Omron CX-Programmer project NewProject (CX-Programmer 9.73)

# PLC NewPLC1: CP1L M

## Global symbols (name address type ; comment)
0.00 BOOL  ; caco
0.01 BOOL  ; box1
0.02 BOOL  ; box2
0.03 BOOL  ; box3
0.04 BOOL  ; box4
0.05 BOOL  ; box5
0.06 BOOL  ; box6
0.07 BOOL  ; reset contagem
0.08 BOOL  ; total peças
0.09 BOOL  ; seleção comercial
D0 CHANNEL  ; contagem box 0
D10 CHANNEL  ; contagem box 5
D12 CHANNEL  ; contagem box 6
D14 CHANNEL  ; contagem total
D18 CHANNEL  ; contador amostragem
D2 CHANNEL  ; contagem box 1
D4 CHANNEL  ; contagem box 2
D6 CHANNEL  ; contagem box 3
D630 CHANNEL  ; Segundos Relógio
D631 CHANNEL  ; Minutos relógio
D632 CHANNEL  ; Horas relógio
D633 CHANNEL  ; Dia relógio
D634 CHANNEL  ; Mes Relógio
D635 CHANNEL  ; Ano relógio
D700 CHANNEL  ; hora ihm
D7003 CHANNEL  ; hora envio
D701 CHANNEL  ; minuto da ihm
D702 CHANNEL  ; segundo ihm
D703 CHANNEL  ; hora do envio
D704 CHANNEL  ; minuto envio
D705 CHANNEL  ; segundo envio
D8 CHANNEL  ; contagem box 4
H10.00 BOOL  ; reset contador
H10.01 BOOL  ; envia relogio
ch400 400 CHANNEL

## Program NewProgram1 (cyclic task 0)
Local symbols
TIM 0.12 BOOL
bit2 BOOL
d400D400 CHANNEL

### Section Controle_Qualidade

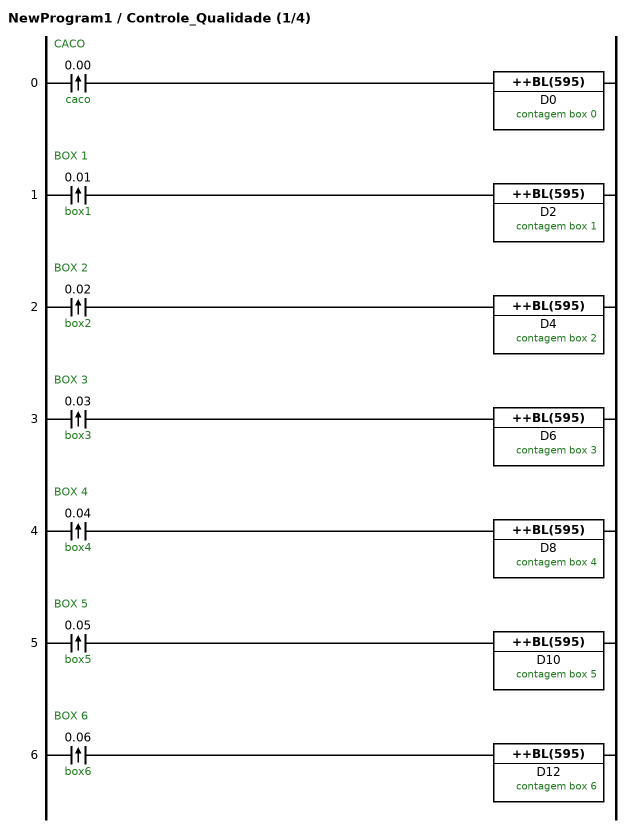
; rung 0: CACO
@LD 0.00  ; caco
++BL(595) D0  ; contagem box 0
; rung 1: BOX 1
@LD 0.01  ; box1
++BL(595) D2  ; contagem box 1
; rung 2: BOX 2
@LD 0.02  ; box2
++BL(595) D4  ; contagem box 2
; rung 3: BOX 3
@LD 0.03  ; box3
++BL(595) D6  ; contagem box 3
; rung 4: BOX 4
@LD 0.04  ; box4
++BL(595) D8  ; contagem box 4
; rung 5: BOX 5
@LD 0.05  ; box5
++BL(595) D10  ; contagem box 5
; rung 6: BOX 6
@LD 0.06  ; box6
++BL(595) D12  ; contagem box 6

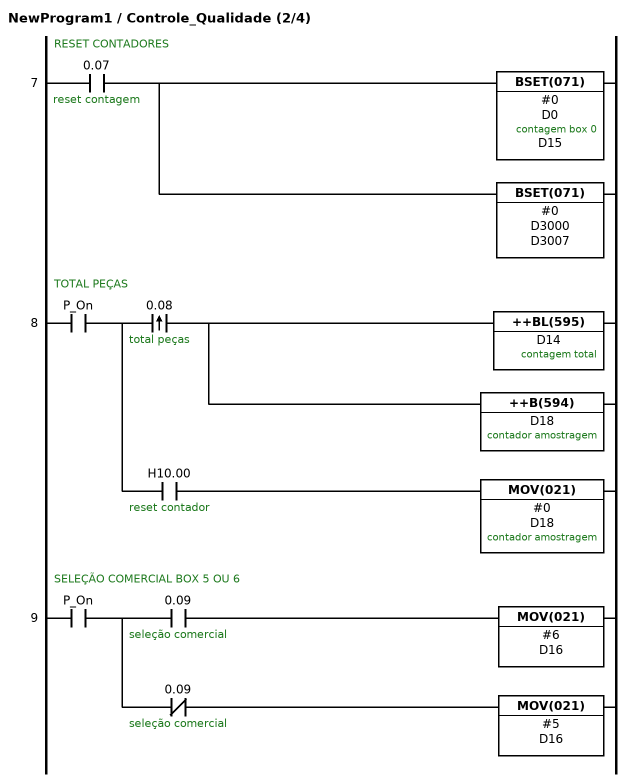
; rung 7: RESET CONTADORES
LD 0.07  ; reset contagem
BSET(071) #0 D0 D15  ; contagem box 0
BSET(071) #0 D3000 D3007
; rung 8: TOTAL PEÇAS
LD P_On
OUT TR0
@AND 0.08  ; total peças
++BL(595) D14  ; contagem total
++B(594) D18  ; contador amostragem
LD TR0
AND H10.00  ; reset contador
MOV(021) #0 D18  ; contador amostragem
; rung 9: SELEÇÃO COMERCIAL BOX 5 OU 6
LD P_On
OUT TR0
AND 0.09  ; seleção comercial
MOV(021) #6 D16
LD TR0
ANDNOT 0.09  ; seleção comercial
MOV(021) #5 D16

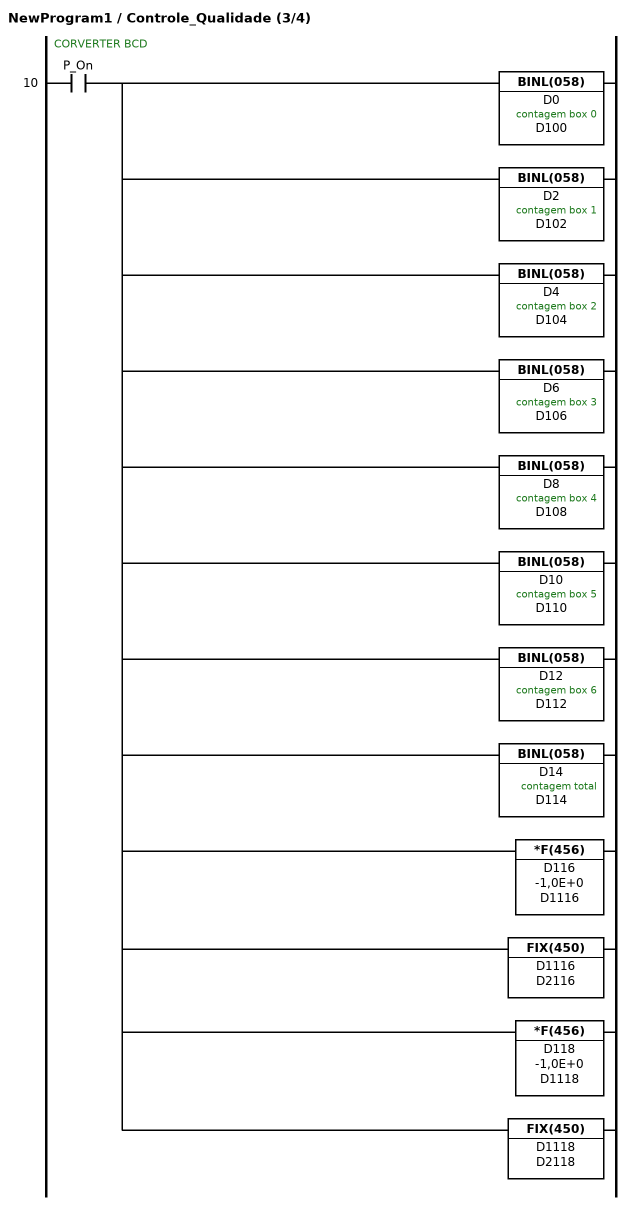
; rung 10: CORVERTER BCD
LD P_On
BINL(058) D0 D100  ; contagem box 0
BINL(058) D2 D102  ; contagem box 1
BINL(058) D4 D104  ; contagem box 2
BINL(058) D6 D106  ; contagem box 3
BINL(058) D8 D108  ; contagem box 4
BINL(058) D10 D110  ; contagem box 5
BINL(058) D12 D112  ; contagem box 6
BINL(058) D14 D114  ; contagem total
*F(456) D116 -1,0E+0 D1116
FIX(450) D1116 D2116
*F(456) D118 -1,0E+0 D1118
FIX(450) D1118 D2118

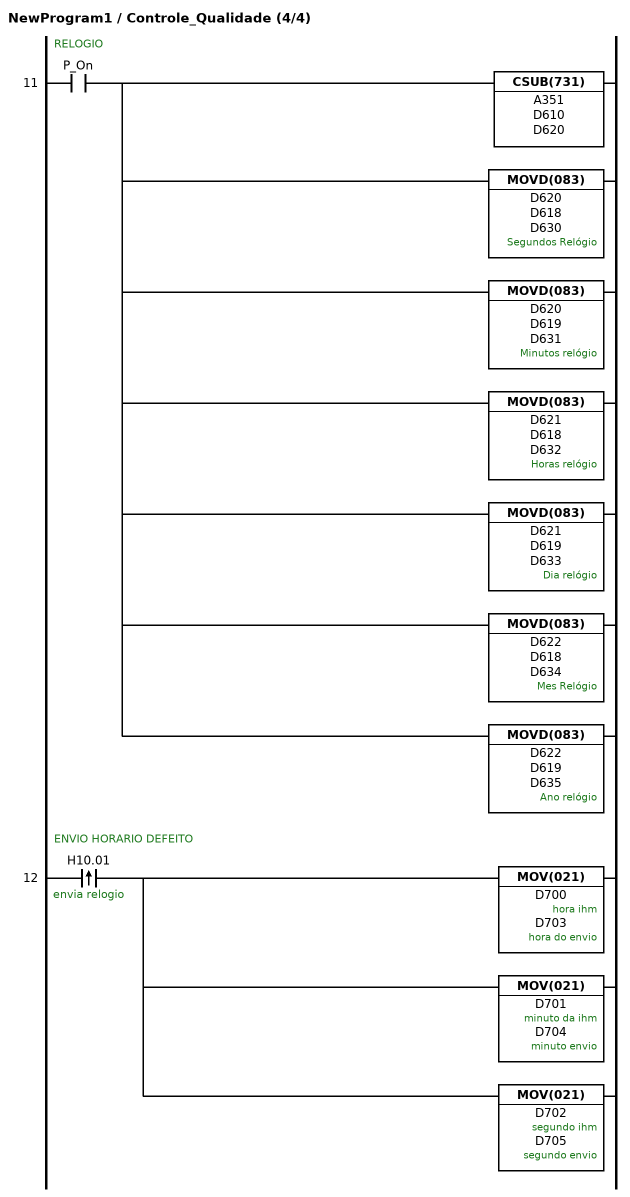
; rung 11: RELOGIO
LD P_On
CSUB(731) A351 D610 D620
MOVD(083) D620 D618 D630  ; Segundos Relógio
MOVD(083) D620 D619 D631  ; Minutos relógio
MOVD(083) D621 D618 D632  ; Horas relógio
MOVD(083) D621 D619 D633  ; Dia relógio
MOVD(083) D622 D618 D634  ; Mes Relógio
MOVD(083) D622 D619 D635  ; Ano relógio
; rung 12: ENVIO HORARIO DEFEITO
@LD H10.01  ; envia relogio
MOV(021) D700 D703  ; hora ihm, hora do envio
MOV(021) D701 D704  ; minuto da ihm, minuto envio
MOV(021) D702 D705  ; segundo ihm, segundo envio

### Section END
; rung 0
END(001)